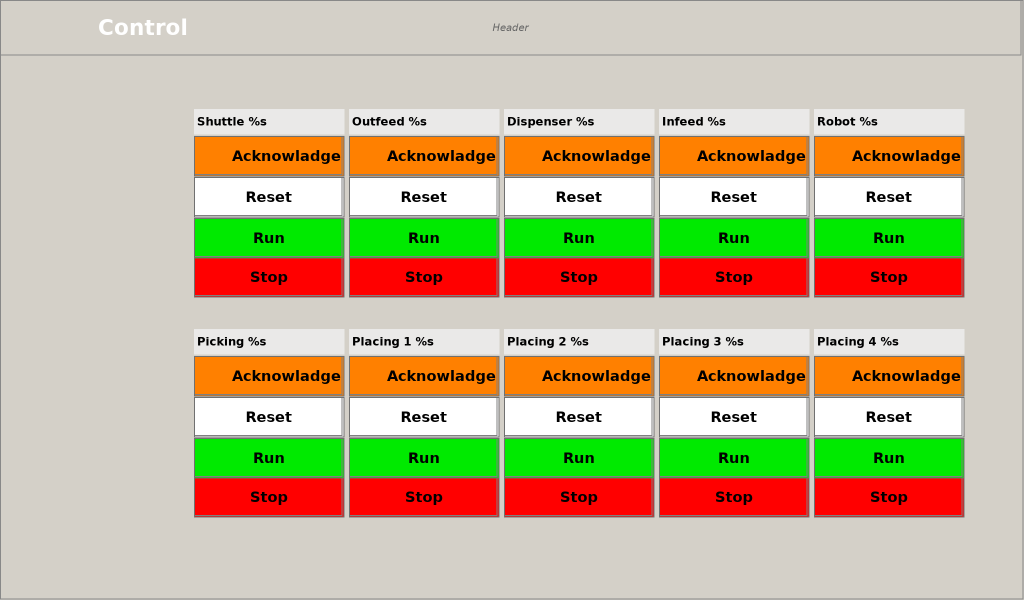
VISUALIZATION StateMachine  // 1024x600
    Frame (0,0 1021x55)
        shows Header()
    Group (194,109 150x188)
        Button (0,27 150x40), "Acknowladge", image: VisuSymbols.Symbols.OK
            tap HMI_GVL.bAcknowledgeButtonShuttle
        Button (0,68 150x40), "Reset", image: VisuSymbols.Symbols.Rec
            tap HMI_GVL.bResetButtonShuttle
        Button (0,148 150x40), "Stop", image: VisuSymbols.Symbols.Stop
            tap HMI_GVL.bStopButtonShuttle
        Button (0,109 150x40), "Run", image: VisuSymbols.Symbols.Play
            tap HMI_GVL.bStartButtonShuttle
        Rectangle (0,0 150x25), "Shuttle %s", text variable: InputOutput_GVL.Shuttle_stsMachine
    Button (349,136 150x40), "Acknowladge", image: VisuSymbols.Symbols.OK
        tap HMI_GVL.bAcknowledgeButtonOutfeed
    Button (349,177 150x40), "Reset", image: VisuSymbols.Symbols.Rec
        tap HMI_GVL.bResetButtonOutfeed
    Button (349,257 150x40), "Stop", image: VisuSymbols.Symbols.Stop
        tap HMI_GVL.bStopButtonOutfeed
    Button (349,218 150x40), "Run", image: VisuSymbols.Symbols.Play
        tap HMI_GVL.bStartButtonOutfeed
    Rectangle (349,109 150x25), "Outfeed %s", text variable: InputOutput_GVL.Outfeed_stsMachine
    Button (504,136 150x40), "Acknowladge", image: VisuSymbols.Symbols.OK
        tap HMI_GVL.bAcknowledgeButtonDispenser
    Button (504,177 150x40), "Reset", image: VisuSymbols.Symbols.Rec
        tap HMI_GVL.bResetButtonDispenser
    Button (504,257 150x40), "Stop", image: VisuSymbols.Symbols.Stop
        tap HMI_GVL.bStopButtonDispenser
    Button (504,218 150x40), "Run", image: VisuSymbols.Symbols.Play
        tap HMI_GVL.bStartButtonDispenser
    Rectangle (504,109 150x25), "Dispenser %s", text variable: InputOutput_GVL.Dispenser_stsMachine
    Group (659,109 150x188)
        Button (0,27 150x40), "Acknowladge", image: VisuSymbols.Symbols.OK
            tap HMI_GVL.bAcknowledgeButtonInfeed
        Button (0,68 150x40), "Reset", image: VisuSymbols.Symbols.Rec
            tap HMI_GVL.bResetButtonInfeed
        Button (0,148 150x40), "Stop", image: VisuSymbols.Symbols.Stop
            tap HMI_GVL.bStopButtonInfeed
        Button (0,109 150x40), "Run", image: VisuSymbols.Symbols.Play
            tap HMI_GVL.bStartButtonInfeed
        Rectangle (0,0 150x25), "Infeed %s", text variable: InputOutput_GVL.Infeed_stsMachine
    Group (814,109 150x188)
        Button (0,27 150x40), "Acknowladge", image: VisuSymbols.Symbols.OK
            tap HMI_GVL.bAcknowledgeButtonRobot
        Button (0,68 150x40), "Reset", image: VisuSymbols.Symbols.Rec
            tap HMI_GVL.bResetButtonRobot
        Button (0,148 150x40), "Stop", image: VisuSymbols.Symbols.Stop
            tap HMI_GVL.bStopButtonRobot
        Button (0,109 150x40), "Run", image: VisuSymbols.Symbols.Play
            tap HMI_GVL.bStartButtonRobot
        Rectangle (0,0 150x25), "Robot %s", text variable: Data_GVL.StateMachineRobot_stsMachine
    Button (194,356 150x40), "Acknowladge", image: VisuSymbols.Symbols.OK
        tap HMI_GVL.bAcknowledgeButtonPicking
    Button (194,397 150x40), "Reset", image: VisuSymbols.Symbols.Rec
        tap HMI_GVL.bResetButtonPicking
    Button (194,477 150x40), "Stop", image: VisuSymbols.Symbols.Stop
        tap HMI_GVL.bStopButtonPicking
    Button (194,438 150x40), "Run", image: VisuSymbols.Symbols.Play
        tap HMI_GVL.bStartButtonPicking
    Rectangle (194,329 150x25), "Picking %s", text variable: Data_GVL.StateMachinePicking_stsMachine
    Button (349,356 150x40), "Acknowladge", image: VisuSymbols.Symbols.OK
        tap HMI_GVL.bAcknowledgeButtonPlacing1
    Button (349,397 150x40), "Reset", image: VisuSymbols.Symbols.Rec
        tap HMI_GVL.bResetButtonPlacing1
    Button (349,477 150x40), "Stop", image: VisuSymbols.Symbols.Stop
        tap HMI_GVL.bStopButtonPlacing1
    Button (349,438 150x40), "Run", image: VisuSymbols.Symbols.Play
        tap HMI_GVL.bStartButtonPlacing1
    Rectangle (349,329 150x25), "Placing 1 %s", text variable: Data_GVL.StateMachinePlacing1_stsMachine
    Button (504,356 150x40), "Acknowladge", image: VisuSymbols.Symbols.OK
        tap HMI_GVL.bAcknowledgeButtonPlacing2
    Button (504,397 150x40), "Reset", image: VisuSymbols.Symbols.Rec
        tap HMI_GVL.bResetButtonPlacing2
    Button (504,477 150x40), "Stop", image: VisuSymbols.Symbols.Stop
        tap HMI_GVL.bStopButtonPlacing2
    Button (504,438 150x40), "Run", image: VisuSymbols.Symbols.Play
        tap HMI_GVL.bStartButtonPlacing2
    Rectangle (504,329 150x25), "Placing 2 %s", text variable: Data_GVL.StateMachinePlacing2_stsMachine
    Button (659,356 150x40), "Acknowladge", image: VisuSymbols.Symbols.OK
        tap HMI_GVL.bAcknowledgeButtonPlacing3
    Button (659,397 150x40), "Reset", image: VisuSymbols.Symbols.Rec
        tap HMI_GVL.bResetButtonPlacing3
    Button (659,477 150x40), "Stop", image: VisuSymbols.Symbols.Stop
        tap HMI_GVL.bStopButtonPlacing3
    Button (659,438 150x40), "Run", image: VisuSymbols.Symbols.Play
        tap HMI_GVL.bStartButtonPlacing3
    Rectangle (659,329 150x25), "Placing 3 %s", text variable: Data_GVL.StateMachinePlacing3_stsMachine
    Button (814,356 150x40), "Acknowladge", image: VisuSymbols.Symbols.OK
        tap HMI_GVL.bAcknowledgeButtonPlacing4
    Button (814,397 150x40), "Reset", image: VisuSymbols.Symbols.Rec
        tap HMI_GVL.bResetButtonPlacing4
    Button (814,477 150x40), "Stop", image: VisuSymbols.Symbols.Stop
        tap HMI_GVL.bStopButtonPlacing4
    Button (814,438 150x40), "Run", image: VisuSymbols.Symbols.Play
        tap HMI_GVL.bStartButtonPlacing4
    Rectangle (814,329 150x25), "Placing 4 %s", text variable: Data_GVL.StateMachinePlacing4_stsMachine
    Label (95,15 214x25), "Control"
END_VISUALIZATION

(* stored: Version 1.1.0.1, ProductVersion 3.1.4024.12
   Visu StateMachine: Id {37f668e3-0daa-4b53-935c-508d501a73df} *)
